FUNCTION WRITE_ANY_DINT : BOOL
VAR_INPUT
    ptr: POINTER TO DINT;
    val: DINT;
END_VAR

ptr^ := val;

END_FUNCTION

(* stored: Version 1.1.0.1, ProductVersion 3.1.4022.9
   POU WRITE_ANY_DINT: Id {e753c22d-5f40-4162-b951-1bab50066302}, SpecialFunc None *)
